FUNCTION_BLOCK EL2022
VAR
	{attribute addProperty Name "WcState"}
	_wcState : WcStateBase;
	{attribute addProperty Name "Info data"}
	_infoData : InfoDataBase;
	_io : EL2xx2_Data;
END_VAR

PROPERTY IO : REFERENCE TO EL2xx2_Data
GET
IO REF= _io;
END_GET
END_PROPERTY

PROPERTY WcState : REFERENCE TO WcStateBase
GET
WcState REF= _wcState;
END_GET
END_PROPERTY

END_FUNCTION_BLOCK

(* stored: Version 1.1.0.1, ProductVersion 3.1.4024.9
   POU EL2022: Id {eed33915-1bdb-09b3-0b02-6b5ca85abc88}, SpecialFunc None
   Property IO: Id {757ff1d0-4e14-0989-095e-95cb17a12ff0}
   Get Get: Id {2e7d38e9-c396-031f-37fe-ee107d3c0c0b}
   Property WcState: Id {1968b3d3-b2dd-0346-36bb-ffd7d0348617}
   Get Get: Id {638e07d5-064b-014d-192b-20c25e5c7ac8} *)
